// TwinCAT 3 PLC project Elevator
// ProgramVersion: 3.1.4023.0
// libraries:
//   Tc2_Standard, * (Beckhoff Automation GmbH)
//   Tc3_Module, * (Beckhoff Automation GmbH)
//   VisuSymbols,3.5.10.0,System
// project tree:
//   Global Vars/ GVL.TcGVL
//   / GlobalTextList.TcGTLO, PlcTask.TcTTO, Visualization Manager.TcVMO (not stored)
//   PRG/ FB_Elevator.TcPOU, FB_Sim.TcPOU, MAIN.TcPOU
//   UDT/ E_States.TcDUT, ST_Floor.TcDUT
//   Visu/ FloorVisu.TcVIS, Visualization.TcVIS
// real-time tasks:
//   TASK PlcTask: cycle T#10ms, priority 20, ADS port 350

CONFIGURATION Elevator
    RESOURCE PLC ON TwinCAT3
        TASK PlcTask(INTERVAL := T#10ms, PRIORITY := 20);
        PROGRAM MAIN WITH PlcTask : MAIN;
    END_RESOURCE
END_CONFIGURATION

// ---- UDT/E_States.TcDUT
{attribute 'qualified_only'}
{attribute 'strict'}
TYPE E_States :
(
	Call := 0,
	MoveUp,
	MoveDown,
	SlowDown,
	Stop
);
END_TYPE

// ---- UDT/ST_Floor.TcDUT
TYPE ST_Floor :
STRUCT
	Call :BOOL;
	High,
	Mid,
	Low :BOOL;
END_STRUCT
END_TYPE

// ---- Global Vars/GVL.TcGVL
VAR_GLOBAL
	Elevator:FB_Elevator;
	Floors:ARRAY[1..4]	OF	ST_Floor;
	RequestedFloor: INT;
	ActualFloor: INT:=1;
	BT_Text:ARRAY[1..4]	OF	STRING:=['Call L1','Call L2','Call L3','Call L4'];
	Elevator_Y:INT;
END_VAR

// ---- PRG/MAIN.TcPOU
PROGRAM MAIN
VAR
	State: E_States;
	i: INT;
	Trigger:ARRAY[1..4]	OF	R_TRIG;
	FB_Sim	:	FB_Sim;
	
	init:BOOL;
END_VAR

IF NOT init THEN
	Floors[1].Mid:=TRUE;
	init:=TRUE;
END_IF

CASE	State	OF
	E_States.Call:
		FOR	i:=1	TO	4	DO
			IF	Floors[i].Call	THEN
				RequestedFloor:=i;
		IF	RequestedFloor>ActualFloor	THEN
			State:=E_States.MoveUp;	
			FB_sim.state:=1;
		ELSIF	RequestedFloor<ActualFloor	THEN
			State:=E_States.MoveDown;	
			FB_sim.state:=16;
		END_IF
			END_IF
		END_FOR
		

	E_States.MoveUp:
		Elevator.MoveUp();
		FOR	i:=1	TO	4	DO
			Trigger[i](clk:=Floors[i].Low);
			IF	Trigger[i].Q	THEN
			//	ActualFloor:=ActualFloor+1;
			END_IF
		END_FOR
		
		IF	ActualFloor=RequestedFloor	THEN
			State:=E_States.SlowDown;
			FB_sim.state:=12;
		END_IF
	E_States.MoveDown:
		Elevator.MoveDown();
		FOR	i:=1	TO	4	DO
			Trigger[i](clk:=Floors[i].High);
			IF	Trigger[i].Q	THEN
			///	ActualFloor:=ActualFloor-1;
			END_IF
		END_FOR
		
		IF	ActualFloor=RequestedFloor	THEN
			State:=E_States.SlowDown;
			FB_sim.state:=27;
		END_IF
		
	E_States.SlowDown:
		Elevator.SlowDown();
		FOR	i:=1	TO	4	DO
			IF	Floors[i].Mid	THEN
				State:=E_States.Stop;
			END_IF
		END_FOR
	E_States.Stop:
		Elevator.Stop();
		State:=E_States.Call;
END_CASE



FB_Sim(Floors:= GVL.Floors, RequestedFloor:= GVL.RequestedFloor, ActualFloor:= GVL.ActualFloor);

END_PROGRAM

// ---- PRG/FB_Sim.TcPOU
FUNCTION_BLOCK FB_Sim
VAR_IN_OUT
	Floors:		ARRAY[1..4]	OF	ST_Floor;
	RequestedFloor: INT;
	ActualFloor: INT;

END_VAR
VAR_INPUT
		state:INT;
END_VAR
VAR

	delay3s	:	TON;
	delay6s	:	TON;
END_VAR

CASE State OF
	1:
		Floors[ActualFloor].Mid:=FALSE;
		state:=State+1;
	2:
		Delay3s.IN:=TRUE;
		IF Delay3s.Q THEN
			state:=state+1;
			Delay3s.IN:=FALSE;
		END_IF
	3:
		GVL.Elevator_Y:=GVL.Elevator_Y-55;
		Floors[ActualFloor].High:=TRUE;
		state:=state+1;
	4:
		Delay3s.IN:=TRUE;
		IF Delay3s.Q THEN
			state:=state+1;
			Delay3s.IN:=FALSE;
		END_IF
	5:
		Floors[ActualFloor].High:=FALSE;
		State:=state+1;
	6:
		Delay6s.IN:=TRUE;
		IF Delay6s.Q THEN
			state:=state+1;
			Delay6s.IN:=FALSE;
			ActualFloor:=ActualFloor+1;
		END_IF
	7:
		GVL.Elevator_Y:=GVL.Elevator_Y-71;
		Floors[ActualFloor].Low:=TRUE;
		state:=state+1;
	8:
		Delay3s.IN:=TRUE;
		IF Delay3s.Q THEN
			state:=state+1;
			Delay3s.IN:=FALSE;
		END_IF
	9:
		Floors[ActualFloor].Low:=FALSE;
		state:=state+1;
	
	10:
		Floors[ActualFloor].Mid:=TRUE;
		state:=state+1;
		GVL.Elevator_Y:=GVL.Elevator_Y-55;
	11:	Delay3s.IN:=TRUE;
		IF Delay3s.Q THEN
			state:=1;
			Delay3s.IN:=FALSE;
		END_IF
	12:
		Floors[ActualFloor].Low:=TRUE;
		state:=state+1;
		GVL.Elevator_Y:=GVL.Elevator_Y-71;
	13:
		Delay3s.IN:=TRUE;
		IF Delay3s.Q THEN
			state:=state+1;
			Delay3s.IN:=FALSE;
		END_IF
	14:
		Floors[ActualFloor].Low:=FALSE;
		state:=state+1;
	15:
		GVL.Elevator_Y:=GVL.Elevator_Y-55;
		Floors[ActualFloor].Low:=FALSE;
		Floors[ActualFloor].High:=FALSE;
		Floors[ActualFloor].Mid:=TRUE;
		state:=99;
		
	16:
		Floors[ActualFloor].Mid:=FALSE;
		State:=State+1;
	17:
		Delay3s.IN:=TRUE;
		IF Delay3s.Q THEN
			state:=state+1;
			Delay3s.IN:=FALSE;
		END_IF
	18:
		Floors[ActualFloor].Low:=TRUE;
		GVL.Elevator_Y:=GVL.Elevator_Y+55;
		state:=state+1;
	
	19:
		Delay3s.IN:=TRUE;
		IF Delay3s.Q THEN
			state:=state+1;
			Delay3s.IN:=FALSE;
		END_IF
	
	20:
		Floors[ActualFloor].Low:=FALSE;
		state:=state+1;
	21:
		Delay6s.IN:=TRUE;
		IF Delay6s.Q THEN
			state:=state+1;
			ActualFloor:=ActualFloor-1;
			
			Delay6s.IN:=FALSE;
		END_IF
	22:
		GVL.Elevator_Y:=GVL.Elevator_Y+71;
		Floors[ActualFloor].High:=TRUE;
		state:=state+1;
	
	23:
		Delay3s.IN:=TRUE;
		IF Delay3s.Q THEN
			state:=state+1;
			Delay3s.IN:=FALSE;
		END_IF
	24:
		Floors[ActualFloor].High:=FALSE;
		GVL.Elevator_Y:=GVL.Elevator_Y+55;
		state:=state+1;
	25:
	Floors[ActualFloor].Mid:=TRUE;
	state:=state+1;	
	
	26:
		Delay3s.IN:=TRUE;
		IF Delay3s.Q THEN
			state:=16;
			Delay3s.IN:=FALSE;
		END_IF
		
	27:
		Floors[ActualFloor].High:=TRUE;
		GVL.Elevator_Y:=GVL.Elevator_Y+71;
		state:=state+1;
	28:
		Delay3s.IN:=TRUE;
		IF Delay3s.Q THEN
			state:=state+1;
			Delay3s.IN:=FALSE;
		END_IF
	29:
		Floors[ActualFloor].High:=FALSE;
		state:=state+1;
	30:
		GVL.Elevator_Y:=GVL.Elevator_Y+55;
		Floors[ActualFloor].Low:=FALSE;
		Floors[ActualFloor].High:=FALSE;
		Floors[ActualFloor].Mid:=TRUE;
		state:=99;	
	
END_CASE

delay3s(IN:= delay3s.IN, PT:= T#500MS, Q=> , ET=> );
delay6s(IN:= delay6s.IN, PT:= T#2S, Q=> , ET=> );

END_FUNCTION_BLOCK

// ---- PRG/FB_Elevator.TcPOU
FUNCTION_BLOCK FB_Elevator
VAR
	Up,
	Down,
	Slow,
	Brake :BOOL;
END_VAR

ACTION MoveDown:
Up:=FALSE;
Down:=TRUE;
Slow:=FALSE;
Brake:=FALSE;
END_ACTION

ACTION MoveUp:
Up:=TRUE;
Down:=FALSE;
Slow:=FALSE;
Brake:=FALSE;
END_ACTION

ACTION SlowDown:
Slow:=TRUE;
END_ACTION

ACTION Stop:
Up:=
Down:=
Slow:=FALSE;
Brake:=TRUE;
END_ACTION

END_FUNCTION_BLOCK

// ---- GlobalTextList.TcGTLO
TEXTLIST GlobalTextList
  302 = '%d'
  481 = '%s'
  685 = 'ActualFloor'
  82 = 'High'
  111 = 'L1 Call'
  985 = 'L2 Call'
  902 = 'L3 Call'
  749 = 'L4 Call'
  651 = 'Low'
  346 = 'Mid'
  487 = 'RequestedFloor'
  930 = 'State'
END_TEXTLIST

// ---- Visu/FloorVisu.TcVIS
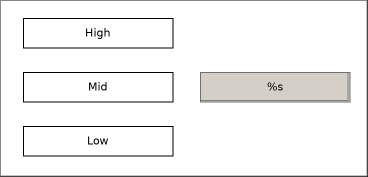
VISUALIZATION FloorVisu  // 368x177
VAR_IN_OUT
	Callbt	:	BOOL;
	Low,Mid,High	:	BOOL;
	name:STRING;
END_VAR
    Rectangle (0,0 368x177)
    Button (200,72 150x30), "%s", text variable: name
        tap Callbt
    Rectangle (23,126 150x30), "Low"
        tap Low
    Rectangle (23,72 150x30), "Mid"
        tap Mid
    Rectangle (23,18 150x30), "High"
        tap High
END_VISUALIZATION

// ---- Visu/Visualization.TcVIS
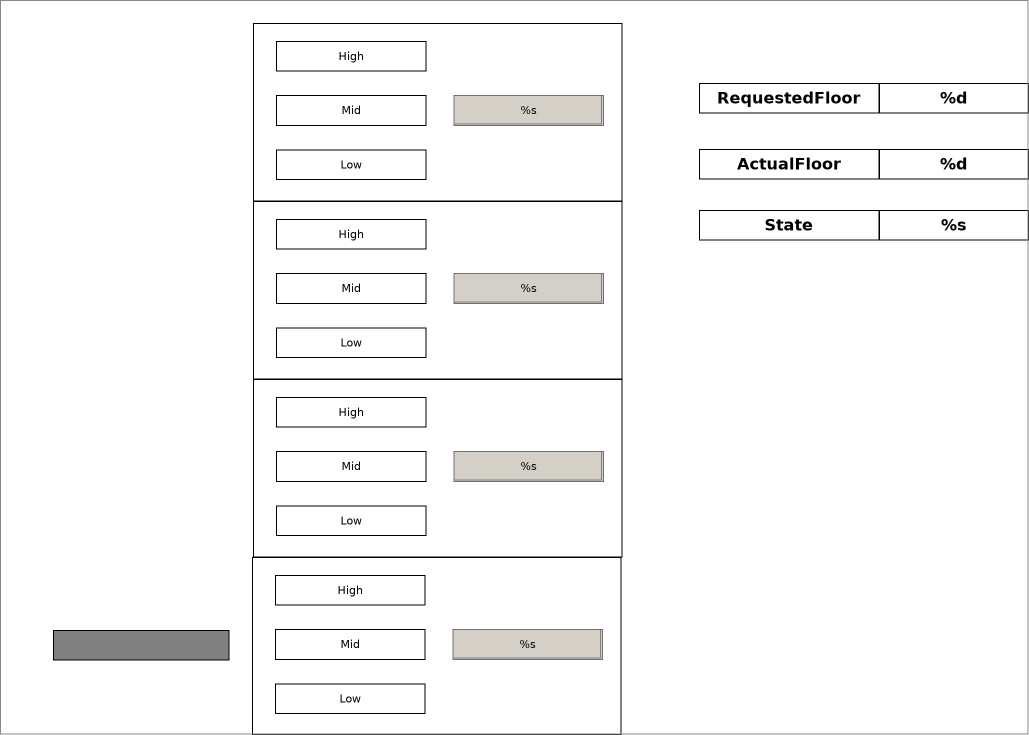
VISUALIZATION Visualization  // 1029x735
    Frame (252,557 369x178)
        shows FloorVisu(Callbt := Floors[1].Call, Low := Floors[1].Low, Mid := Floors[1].mid, High := Floors[1].High, name := BT_Text[1])
    Frame (253,379 369x178)
        shows FloorVisu(Callbt := Floors[2].Call, Low := Floors[2].Low, Mid := Floors[2].Mid, High := Floors[2].High, name := BT_Text[2])
    Frame (253,201 369x178)
        shows FloorVisu(Callbt := Floors[3].Call, Low := Floors[3].Low, Mid := Floors[3].Mid, High := Floors[3].High, name := BT_Text[3])
    Frame (253,23 369x178)
        shows FloorVisu(Callbt := Floors[4].Call, Low := Floors[4].Low, Mid := Floors[4].Mid, High := Floors[4].High, name := BT_Text[4])
    Rectangle (699,83 180x30), "RequestedFloor"
    Rectangle (699,149 180x30), "ActualFloor"
    Rectangle (879,83 150x30), "%d", text variable: RequestedFloor
    Rectangle (879,149 150x30), "%d", text variable: ActualFloor
    Rectangle (699,210 180x30), "State"
    Rectangle (879,210 150x30), "%s", text variable: MAIN.State
    Rectangle (53,630 176x30)
        p2738717112: Elevator_Y
END_VISUALIZATION
